FUNCTION F_NOW_MONOTONIC (* returns current monotonic clock value *)
  PACKAGE eclipse4diac::utils::timing;
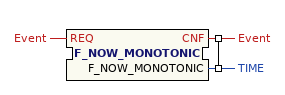
  EVENT_INPUT
    REQ;
  END_EVENT
  EVENT_OUTPUT
    CNF WITH F_NOW_MONOTONIC;
  END_EVENT
  VAR_OUTPUT
    F_NOW_MONOTONIC : TIME;
  END_VAR
  BODY IN ST:
PACKAGE utils::timing;

(* returns current monotonic clock value *)
FUNCTION F_NOW_MONOTONIC : TIME
F_NOW_MONOTONIC := NOW_MONOTONIC();
END_FUNCTION
  END_BODY
END_FUNCTION
